{region '#Template'}
	{attribute 'Version' := '1.0.0.0'}
	{attribute 'Tags' := '"LCID": "1031", "Text": "Universal, Control, Antiblockierschutz"'}
	{attribute 'Tags' := '"LCID": "1033", "Text": "Universal, Control, Anti-blocking protection"'}
	{attribute 'Description' := '"LCID": "1031", "Text": "Antiblockierschutz"'}
	{attribute 'Description' := '"LCID": "1033", "Text": "Anti-blocking protection"'}
{endregion}
FUNCTION_BLOCK FB_BA_AntiBlocking EXTENDS FB_BA_View
VAR_INPUT
	bFdb					: BOOL;	
	bExtReq					: BOOL;
	bLock					: BOOL;
END_VAR
VAR_OUTPUT
	bQ						: BOOL;
END_VAR
VAR_INPUT CONSTANT PERSISTENT
	{attribute 'parameterCategory' := 'Operation'}
	bEn : BOOL := TRUE;
END_VAR
VAR_INPUT CONSTANT
	IdlePrd					: FB_BA_AV_Op;									 
	ImpulseLength			: FB_BA_AV_Op;
END_VAR	
VAR		
	AblkFnct				: FB_BA_AntBlkg;
	tonEn					: TON;
END_VAR

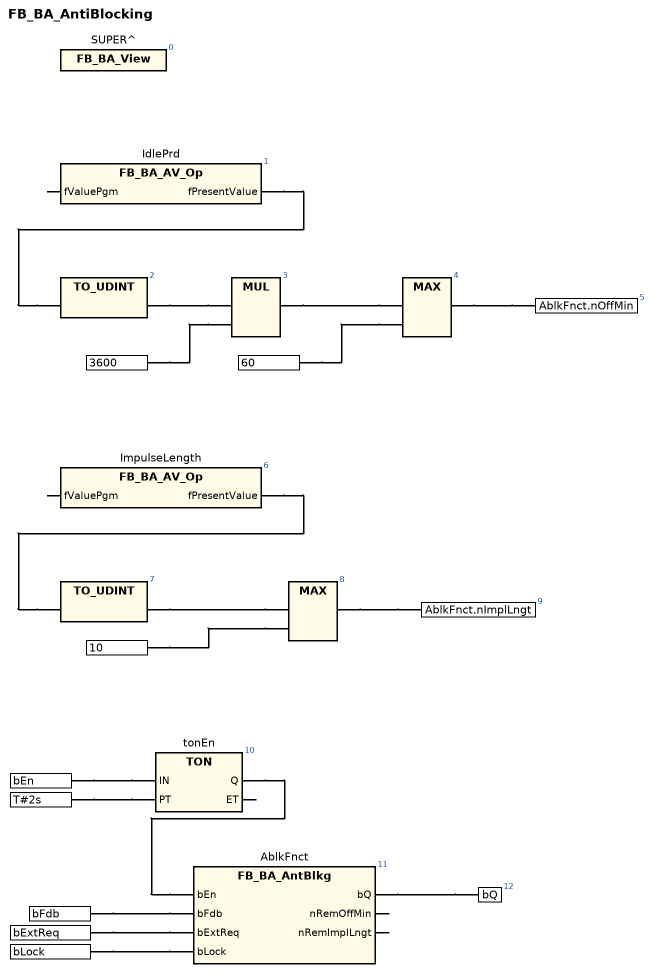
SUPER^(); // FB_BA_View
IdlePrd(); // FB_BA_AV_Op
AblkFnct.nOffMin := MAX(TO_UDINT(IdlePrd.fPresentValue) * 3600, 60);
ImpulseLength(); // FB_BA_AV_Op
AblkFnct.nImplLngt := MAX(TO_UDINT(ImpulseLength.fPresentValue), 10);
tonEn(IN := bEn, PT := T#2s); // TON
AblkFnct(bEn := tonEn.Q, bFdb := bFdb, bExtReq := bExtReq, bLock := bLock); // FB_BA_AntBlkg
bQ := AblkFnct.bQ;

METHOD FB_init : BOOL
VAR_INPUT
	bInitRetains : BOOL; // if TRUE, the retain variables are initialized (warm start / cold start)
	bInCopyCode : BOOL;  // if TRUE, the instance afterwards gets moved into the copy code (online change)
END_VAR
IdlePrd.iParent					:= THIS^;
IdlePrd.iLabel					:= LblUniControl.AntiBlocking_IdlePeriod;	
IdlePrd.sObjectName				:= '{Idx=01}';								 	 
IdlePrd.eUnit 					:= E_BA_Unit.eTime_Hours;								 
IdlePrd.fValueRm				:= 168;
IdlePrd.fCOVIncrement			:= BA2_Param.fDefCOVIncrement;
														 
ImpulseLength.iParent			:= THIS^;
ImpulseLength.iLabel			:= LblUniControl.AntiBlocking_ImpulsLength;	
ImpulseLength.sObjectName		:= '{Idx=01}';								 	 
ImpulseLength.eUnit 			:= E_BA_Unit.eTime_Seconds;								 
ImpulseLength.fValueRm			:= 240;					
ImpulseLength.fCOVIncrement		:= BA2_Param.fDefCOVIncrement;
END_METHOD

END_FUNCTION_BLOCK

(* stored: Version 1.1.0.1, ProductVersion 3.1.4024.9
   POU FB_BA_AntiBlocking: Id {3290d95b-bb6e-4b6e-a6f1-68b7f02c36c0}, SpecialFunc None
   Method FB_init: Id {3b79f36a-6e98-4304-838e-9c5daec17070} *)
